TEXTLIST TextListXPIMStates
  0 = 'Unknown'
  1 = 'Out'
  2 = 'Yag'
  3 = 'Diamond'
  4 = 'Reticle'
   = ''
END_TEXTLIST

(* stored: Version 1.1.0.1, ProductVersion 3.1.4022.18
   TextList TextListXPIMStates: Id {c824132c-c8ae-46d7-805b-cf1e1aee9301} *)
